{attribute 'qualified_only'}
VAR_GLOBAL
	stEnable : ST_Enabeling; 
END_VAR

(* stored: Version 1.1.0.1, ProductVersion 3.1.4024.12
   GVL GVL_HMIvars: Id {5580be2b-47fe-45e8-83de-72f2598e6fc0} *)
